(*			
	RAFALOS
	Rafał Osajda		23.09.2025		TC 4024.66
	Struktura pomocnicza potrzeba do wiazania zmiennych
*)
TYPE ST_BaseGroupElement_HMI_Link :
STRUCT
	stBaseLoggerElement				: ST_BaseLoggerElement_HMI;
	stBaseComponent					: ST_BaseComponent_HMI;
	stBaseControlElement			: ST_BaseControlElement_HMI;
	stBaseGroupElement				: ST_BaseGroupElement_HMI;
END_STRUCT
END_TYPE

(* stored: Version 1.1.0.1
   DUT ST_BaseGroupElement_HMI_Link: Id {74a7ec16-ee53-0f43-0990-47b1e1031fb1} *)
